// TIA Portal V19 export
TYPE "NetworkSwitchHMI"
   STRUCT
      Ports { S7_SetPoint := 'True'} : Array[1..8] of "LPNDR_typePortInformation";
      Port { S7_SetPoint := 'True'} : "LPNDR_typePortInformation";
      Index { S7_SetPoint := 'True'} : Int := 1;
   END_STRUCT;
END_TYPE
